PROGRAM Math
VAR
END_VAR

METHOD AddInt : INT
VAR_INPUT
  a : INT;
  b : INT;
END_VAR
AddInt := a + b;
END_METHOD

END_PROGRAM

(* stored: Version 1.1.0.1, ProductVersion 3.1.4026.12
   POU Math: Id {53549243-095a-493a-ab32-c0c5bbf86db2}, SpecialFunc None
   Method AddInt: Id {a7dbd43a-20a6-4288-80d8-5bcf4f8bfa94} *)
